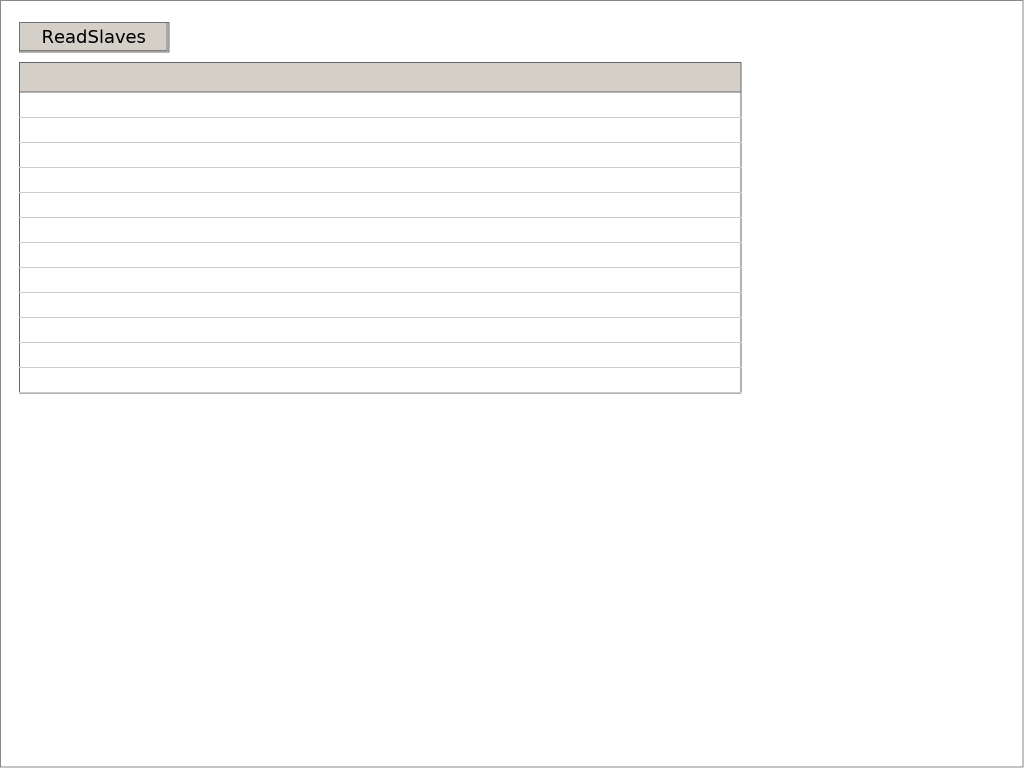
VISUALIZATION Visualization  // 1024x768
    Button (19,22 150x30), "ReadSlaves"
        tap prgECatDiag.bGetStates
    Table (19,62 722x331), data array: prgECatDiag.aSlaveInfo
        p1014161805: PRGECATDIAG.cMaxNumOfSlaves - 0 + INT#1
        p3854506369: prgECatDiag.aSlaveInfo[INDEX].configDevName
        p1892666644: prgECatDiag.aSlaveInfo[INDEX].scannedDevName
        p338671338: prgECatDiag.aSlaveInfo[INDEX].addr
        p2170511999: prgECatDiag.aSlaveInfo[INDEX].devState
        p511219082: Nome escaneado
        p1755163831: Endereço
        p4092479075: Estado
END_VISUALIZATION

(* stored: Version 1.1.0.1
   Visu Visualization: Id {fe2538c0-3240-49b4-b9c2-e225a1ad0371} *)
